(* PLC project CoDeSys External Library Template, WAGO e!COCKPIT e!COCKPIT, author 3S - Smart Software Solutions GmbH *)
(* stored: creationDateTime 2019-10-29T12:37:19.4247485, version 3.5.5.30, modificationDateTime 2019-10-29T12:36:39.3744516, organization 3S - Smart Software Solutions GmbH *)
(* Library project template with all possible element types, docu and a sample project structure *)

(* values of enumPPPSSilownikSABpError: BrakKomunikacji: brak komunikacji (po EnOcean) z siłownikiem; AlarmOgolny: alarm ogólny; DetekcjaOtwarciaOkna: błąd baterii; Defrost: defrost; AlarmCzujnika: alarm braku zmiany wartości czujnika temp. *)

(* Autor: Paweł Kąkol, 2018-09-04-PK Prawa majątkowe: Solwena Sp. z o.o., Aktualizacje: 2019-01-28-JC - defrost 2019-02-14-AWy - alarm czujnika temperatury Opis: enum służy do obsługi alarmów w fb siłownika (SAB+) HRU0 na budynkach PPP Sopot *)
{attribute 'qualified_only'}
{attribute 'strict'}
TYPE enumPPPSSilownikSABpError : (BrakKomunikacji := 1, AlarmOgolny := 2, DetekcjaOtwarciaOkna := 3, Defrost := 4, AlarmCzujnika := 5);
END_TYPE
